Staubli VAL3: renameFile.pgx

program renameFile()
  local bool l_bRes
begin
  //rename file or folder
  l_bRes=$rename(sFromRename,sToRename)
  if l_bRes
    gotoxy(1,5)
    put("更名："+sFromRename+"至"+sToRename)
  else
    gotoxy(1,5)
    put("更名失败："+sFromRename+"至"+sToRename)
  endIf
end
